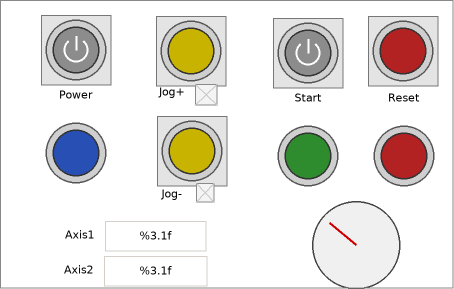
VISUALIZATION Visualization  // 454x289
    Lamp1 (41,118 70x70), variable: MAIN.bAllAxisPowerOn, style: Lamp-Lamp1-Blue
    PowerSwitch (41,15 70x70), variable: MAIN.bPower, behaviour: TOGGLE, style: Switch-PowerSwitch-Gray
    Label (26,80 100x30), "Power"
    PushSwitch (156,16 70x70), variable: MAIN.bJogPlus, behaviour: TAP, style: Switch-PushSwitch-Yellow
    Label (122,77 100x30), "Jog+"
    Label (122,179 100x30), "Jog-"
    PushSwitch (157,116 70x70), variable: MAIN.bJogMinus, behaviour: TAP, style: Switch-PushSwitch-Yellow
    PowerSwitch (273,18 70x70), variable: MAIN.bStart, behaviour: TOGGLE, style: Switch-PowerSwitch-Gray
    Lamp1 (273,121 70x70), variable: MAIN.bStart, style: Lamp-Lamp1-Green
    Label (258,83 100x30), "Start"
    Lamp1 (369,121 70x70), variable: MAIN.bError, style: Lamp-Lamp1-Red
    Label (354,83 100x30), "Reset"
    PushSwitch (368,16 70x70), variable: MAIN.bReset, behaviour: TOGGLE, style: Switch-PushSwitch-Red
    Textfield (105,221 101x30), "%3.1f", text variable: MAIN.stAxis1.NcToPlc.ActPos
    Label (47,220 66x30), "Axis1"
    Label (46,255 66x30), "Axis2"
    Textfield (104,256 103x30), "%3.1f", text variable: MAIN.stAxis2.NcToPlc.ActPos
    Image (195,84 22x21), image: VisuSymbols.Symbols.ArrowHalfLeftLeft
    Image (196,183 18x19), image: VisuSymbols.Symbols.ArrowHalfRightDown
    Meter180 (259,201 194x88), value: MAIN.stAxis1.NcToPlc.ActVelo, style: Meter-Meter180-Blue, scale format: %.1f, scale -1000..1000
END_VISUALIZATION

(* stored: Version 1.1.0.1, ProductVersion 3.1.4024.11
   Visu Visualization: Id {fd48ea7b-7c45-4554-bf2d-93f8b2384732} *)
